{attribute 'linkalways'} 
{attribute 'no_explicit_call' := 'This FB is a CLASS and must be accessed using methods or properties'}
{attribute 'enable_dynamic_creation'}
FUNCTION_BLOCK FINAL ABS_REAL EXTENDS Node
VAR
	in : _REAL(0.0);
	out : _REAL(0.0);
END_VAR

METHOD PUBLIC Clone : I_Node
VAR
	pNode : POINTER TO ABS_REAL;
END_VAR
pNode := __NEW(ABS_REAL);
Clone := pNode^;
END_METHOD

METHOD FB_init : BOOL
VAR_INPUT
	bInitRetains : BOOL; // if TRUE, the retain variables are initialized (warm start / cold start)
	bInCopyCode : BOOL;  // if TRUE, the instance afterwards gets moved into the copy code (online change)
END_VAR
AddInput('in',THIS^.in);
AddOutput('out', THIS^.out);
END_METHOD

METHOD PROTECTED OnExecute
VAR
END_VAR
out.Value := ABS(in.Value);
END_METHOD

END_FUNCTION_BLOCK

(* stored: Version 1.1.0.1, ProductVersion 3.1.4024.15
   POU ABS_REAL: Id {01acfcd9-8374-4d03-85c1-d771abc6a4fe}, SpecialFunc None
   Folder Constructor: Id {908253e0-412c-498e-b36f-506d810b47f0}
   Method Clone: Id {ee85025b-911a-487f-ac04-cef345320cf5}
   Method FB_init: Id {3f01b689-ab47-42ee-901d-ec9510342cc4}
   Method OnExecute: Id {ca6f1d4e-1da7-4ee4-b838-7ddce2e404db} *)
